// TIA Portal V17 export
// export: Created 2023-11-01T05:26:42.6428423Z, ExportSetting WithDefaults, DisplayName Totally Integrated Automation Portal, DisplayVersion V17, DisplayName TIA Portal Openness, DisplayVersion V17, DisplayName TIA Portal Version Control Interface, DisplayVersion V17, DisplayName STEP 7 Professional, DisplayVersion V17, DisplayName STEP 7 Safety, DisplayVersion V17, DisplayName WinCC Professional, DisplayVersion V17
VAR_GLOBAL   // PLC tag table "Default tag table"
   Tag_1 AT %I0.0 : Bool;
   Tag_2 AT %Q0.0 : Bool;
   Tag_3 AT %I0.1 : Bool;
END_VAR
